// TIA Portal V19 program export: 0 tag tables, 0 data types, 1 data blocks, 2 code blocks (in call order from the OBs), 0 instance data blocks

DATA_BLOCK "ceD"   // DB1
{ S7_Optimized_Access := 'TRUE' }
VERSION : 0.1
// stored: AutoNumber true, DBAccessibleFromOPCUA true, DBAccessibleFromWebserver true, IsOnlyStoredInLoadMemory false, IsRetainMemResEnabled false, IsWriteProtectedInAS false, MemoryReserve 100
   VAR
      IN : Struct
         in1 : Bool;
         in2 : Int;
         in3 : Int;
         in4 : Int;
         in5 : Bool;
      END_STRUCT;
      out : Struct
         out1 : Bool;
         out2 : Int;
         out3 : Int;
      END_STRUCT;
   END_VAR
BEGIN
END_DATA_BLOCK

ORGANIZATION_BLOCK "Main"   // OB1, LAD, ProgramCycle
TITLE = "Main Program Sweep (Cycle)"
{ S7_Optimized_Access := 'TRUE' }
VERSION : 0.1
// stored: AutoNumber true, IsIECCheckEnabled false, SetENOAutomatically false
   VAR_INPUT
      Initial_Call : Bool;
      Remanence : Bool;
   END_VAR
BEGIN

REGION Network 1
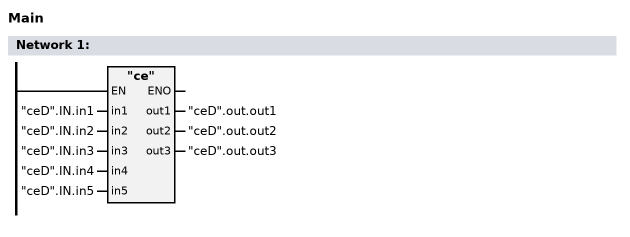
   RUNG wire#powerrail
      "ce"(in1 := "ceD".IN.in1, in2 := "ceD".IN.in2, in3 := "ceD".IN.in3, in5 := "ceD".IN.in5, in4 := "ceD".IN.in4, out1 => "ceD".out.out1, out2 => "ceD".out.out2, out3 => "ceD".out.out3)
   END_RUNG
   // the same network as SCL:
   "ce"(in1 := "ceD".IN.in1,
        in2 := "ceD".IN.in2,
        in3 := "ceD".IN.in3,
        in4 := "ceD".IN.in4,
        in5 := "ceD".IN.in5,
        out1 => "ceD".out.out1,
        out2 => "ceD".out.out2,
        out3 => "ceD".out.out3);
END_REGION
END_ORGANIZATION_BLOCK

FUNCTION "ce" : Void   // FC1, LAD
{ S7_Optimized_Access := 'TRUE' }
VERSION : 0.1
// stored: AutoNumber true, IsIECCheckEnabled false, SetENOAutomatically false, UDAEnableTagReadback false
   VAR_INPUT
      in1 : Bool;
      in2 : Int;
      in3 : Int;
      in4 : Int;
      in5 : Bool;
   END_VAR
   VAR_OUTPUT
      out1 : Bool;
      out2 : Int;
      out3 : Int;
   END_VAR
BEGIN

REGION Network 1
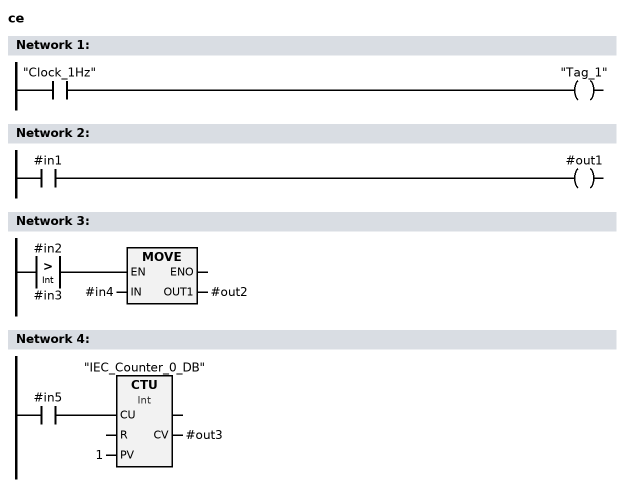
   RUNG wire#powerrail
      Contact( "Clock_1Hz" )
      Coil( "Tag_1" )
   END_RUNG
   // the same network as SCL:
   "Tag_1" := "Clock_1Hz";
END_REGION

REGION Network 2
   RUNG wire#powerrail
      Contact( #in1 )
      Coil( #out1 )
   END_RUNG
   // the same network as SCL:
   #out1 := #in1;
END_REGION

REGION Network 3
   RUNG wire#powerrail
      { S7_Templates := "SrcType := Int" } GT_Contact(in1 := #in2, in2 := #in3)
      Move(in := #in4, out1 => #out2)
   END_RUNG
   // the same network as SCL:
   IF #in2 > #in3 THEN #out2 := #in4; END_IF;
END_REGION

REGION Network 4
   RUNG wire#powerrail
      Contact( #in5 )
      { S7_Templates := "value_type := Int" } "IEC_Counter_0_DB".CTU(r :=, pv := 1, cv => #out3)
   END_RUNG
   // the same network as SCL:
   "IEC_Counter_0_DB".CTU(CU := #in5, PV := 1, CV => #out3);
END_REGION
END_FUNCTION
